TYPE ST_PNOutput_DCExpansion :
STRUCT
	statusbits	: DWORD;
	Busvoltage	: DWORD;
	RatedPower	: DWORD;
	LoadPercentage	: DWORD;
	CurrentPower	: DWORD;
END_STRUCT
END_TYPE

(* stored: Version 1.1.0.1, ProductVersion 3.1.4024.12
   DUT ST_PNOutput_DCExpansion: Id {2322b0d6-524e-42fe-9ddc-636380dcc084} *)
